INTERFACE itfScale

METHOD mScale : INT
VAR_INPUT
END_VAR
END_METHOD

PROPERTY pAnalogSignal : INT
GET
END_GET
SET
END_SET
END_PROPERTY

PROPERTY pMaxSignalValue : INT
GET
END_GET
SET
END_SET
END_PROPERTY

PROPERTY pMaxUnitValue : INT
GET
END_GET
SET
END_SET
END_PROPERTY

PROPERTY pScaledSignal : INT
GET
END_GET
SET
END_SET
END_PROPERTY

END_INTERFACE

(* stored: Version 1.1.0.1, ProductVersion 3.1.4024.12
   Itf itfScale: Id {dde49b6b-a7ba-4a12-8bdd-e88ae290e95f}
   Method mScale: Id {b8b034f4-be24-470c-9904-5df46717c742}
   Property pAnalogSignal: Id {2b180f88-25ae-4af5-b831-0b2d77ff24d5}
   Get Get: Id {e9e69682-c556-4fa0-92b4-9762709e6040}
   Set Set: Id {dd4d643d-a3aa-4343-9dc2-0bce8b1d96e0}
   Property pMaxSignalValue: Id {29a7785c-73ef-4992-a140-a9f8bc24bc0e}
   Get Get: Id {4e594e15-cac1-424d-8e96-fe4170a64aa3}
   Set Set: Id {a6838618-e2f7-406a-9e1f-1ced1df38344}
   Property pMaxUnitValue: Id {05a02cc9-6753-4eeb-b32d-4b8e79fc4c0c}
   Get Get: Id {cf7cb978-66d8-42f7-973c-c6db4faeff04}
   Set Set: Id {d9df3410-9177-4bd5-8531-277217d38c54}
   Property pScaledSignal: Id {c24106c5-7153-44d8-9d0f-3faffabfaabd}
   Get Get: Id {c7f59130-986a-46a6-9334-44837a2cbf88}
   Set Set: Id {b350ad28-7e31-4242-827a-533d102870c4} *)
